{attribute 'GeneratedUsingTerminal: EL5151-0000-0020'}
{attribute addProperty BoxType "EL5151-0000-0020"}
{attribute addProperty Id "StatusAT %I*Status_3E6F3FF310Counter_valueAT %I*UINT2Latch_valueAT %I*UINT2"}
{attribute addProperty CRC "3008586885"}
{attribute addProperty Size "14"}
TYPE ENC_Inputs_B3536485 :
STRUCT
	{attribute addProperty Name "Status"}
	Status AT %I* : Status_3E6F3FF3;
	{attribute addProperty Name "Counter_value"}
	Counter_value AT %I* : UINT;
	{attribute addProperty Name "Latch_value"}
	Latch_value AT %I* : UINT;
END_STRUCT
END_TYPE

(* stored: Version 1.2.0.0, ProductVersion 3.1.4024.9
   DUT ENC_Inputs_B3536485: Id {21de98fe-8967-452c-8ce1-52d35e0d29c0} *)
